Fanuc KAREL source: kd00034.KL

-- PROVISIONAL review KL for V770-1; original PC SHA256 5a4b046a41d9388f735e4f637589a9f03273aa202dfe67c9e77e68be5b13c1d2
-- Incomplete behavior may be omitted. Consult companion uncertainty JSON. Do not deploy.
PROGRAM KD00034
%NOLOCKGROUP
VAR
  I : INTEGER
  J : INTEGER
  B : BOOLEAN
  R : REAL
  S : STRING[80]
BEGIN
  -- UNRESOLVED_PC offsets 5-27; opcodes 9D,81,18,22,9D,12,22,9D,13,04
  -- UNRESOLVED_PC offsets 32-36; opcodes 7F
END KD00034
